# B&R Automation Studio project prjAxis
Automation Studio 6.0.1.7; technology packages: mappMotion 6.0.437033, OpcUaCs 6.0.0

## Configuration Config1

CPU X20CP1686X, AutomationRuntime 6.0.0, Build 11.3.0, Safety 0.0, Vc 6.0.1

### Task classes (Cpu.sw)
```
Cyclic#1 (cycle 2000 us, tolerance 0 us):
  Program <- Program.prg
DataObjects: McAcpSys
NcDataObjects: Capping <- Capping.dob, McDriveLog
Binaries: arsvcreg, udbdef, McAcpDrv, arflatprv, arcoal, FWRules, TCData, McAcpSim, ashwd, Config_1, ashwac, User, sysconf, asfw, arconfig, iomap, Config_3, Config_2, Role
Libraries: runtime, asieccon, powerlnk, astime, fileio, asepl, sys_lib, McBase, MpBase, McAcpAx, McAxis, MpAxis
```

### Hardware
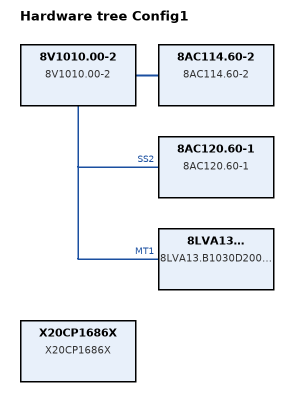
```
8AC114.60-2 : 8AC114.60-2 v2.2.0.0 (NodeNumber=1)  [SS -> 8V1010.00-2.SS1; PLK1 -> X20CP1686X.IF3 [Cable Type=PowerlinkCable, Length=10, Version=1.0.0.3]]
8AC120.60-1 : 8AC120.60-1 v2.2.0.0  [SS -> 8V1010.00-2.SS2]
  PlugInType = Encoder
  McAcoposTypeID = AcoposPlugInConfig
8LVA13.B1030D200-0 : 8LVA13.B1030D200-0 v2.2.0.4  [MT -> 8V1010.00-2.MT1]
  M1/MotorParameters:
    MOTOR_AMB_TEMP_RATED = 40
8V1010.00-2 : 8V1010.00-2 v2.3.0.1
  DriveConfiguration/Module:
    McAcoposTypeID = AcoposConfig
    ActivateACOPOSSimulationOnPLC = 0
    PowerSupply = ETA
  DriveConfiguration/Channel[1]/RealAxis:
    AxisReference = gAxisMaster
    MechanicalElementsIsInvisible = 0
  DriveConfiguration/Channel[1]/RealAxis/MechanicalElements/Gearbox:
    InputIsReadOnly = 0
    Input = 1
    OutputIsReadOnly = 0
    Output = 1
  DriveConfiguration/Channel[1]/RealAxis/MechanicalElements/RotaryToLinearTransformation:
    ReferenceDistanceIsReadOnly = 0
    ReferenceDistance = 1
  DriveConfiguration/Channel[1]/RealAxis/Controller:
    ModeIsReadOnly = 0
    Mode = PositionController
  DriveConfiguration/Channel[1]/RealAxis/Controller/Mode/Position:
    ProportionalGain = 50.0
    IntegrationTime = 0.0
    PredictionTime = 0.0004
    TotalDelayTime = 0.0004
  DriveConfiguration/Channel[1]/RealAxis/Controller/Mode/Speed:
    ProportionalGainIsReadOnly = 0
    ProportionalGain = 2.0
    IntegrationTimeIsReadOnly = 0
    IntegrationTime = 0.0
    FilterTimeIsReadOnly = 0
    FilterTime = 0.0
  DriveConfiguration/Channel[1]/RealAxis/Controller/Mode/LoopFilters:
    LoopFilterXIsReadOnly = 0
    LoopFilter1 = NotUsed
    LoopFilter2 = NotUsed
    LoopFilter3 = NotUsed
  DriveConfiguration/Channel[1]/RealAxis/Homing:
    ModeIsReadOnly = 0
    Mode = Direct
  DriveConfiguration/Channel[1]/RealAxis/Homing/Mode:
    Position = 0.0
    ReferencePulse = NotUsed
  DriveConfiguration/Channel[1]/RealAxis/Homing:
    RestorePositionVariable = 
  DriveConfiguration/Channel[1]/RealAxis/StopReaction:
    QuickstopIsReadOnly = 0
    Quickstop = DecelerationLimit
    DriveErrorIsReadOnly = 0
    DriveError = DecelerationLimit
  DriveConfiguration/Channel[1]/RealAxis/MovementErrorLimits:
    PositionError = 10.0
    VelocityErrorMonitoring = Automatic1
  DriveConfiguration/Channel[1]/RealAxis:
    JerkFilterIsReadOnly = 0
    JerkFilter = NotUsed
    ZeroVibrationFilter = NotUsed
  DriveConfiguration/Channel[1]/RealAxis/DigitalInputs/HomingSwitch:
    SourceIsReadOnly = 0
    Source = X1Ref
    Level = High
  DriveConfiguration/Channel[1]/RealAxis/DigitalInputs/PositiveLimitSwitch:
    Source = X1PosLim
    Level = High
  DriveConfiguration/Channel[1]/RealAxis/DigitalInputs/NegativeLimitSwitch:
    Source = X1NegLim
    Level = High
  DriveConfiguration/Channel[1]/RealAxis/DigitalInputs/Trigger1:
    Source = X1Trigger1
    Level = High
  DriveConfiguration/Channel[1]/RealAxis/DigitalInputs/Trigger2:
    Source = X1Trigger2
    Level = High
  DriveConfiguration/Channel[1]/RealAxis/DigitalInputs/Quickstop:
    Input = Trigger2
  DriveConfiguration/Channel[1]/RealAxis/Simulation:
    SimulationModeOnPLC = CompleteControlledSystem
  DriveConfiguration/Channel[1]/RealAxis/Simulation/SimulationModeOnPLC:
    LoadModel = OneMassBasedOnMotorParameters
  DriveConfiguration/Channel[1]/RealAxis/Simulation/SimulationModeOnPLC/LoadModel:
    AdditiveLoadParID = 0
  DriveConfiguration/Channel[1]/RealAxis/Simulation:
    SimulationModeOnACOPOS = NotUsed
  DriveConfiguration/Channel[1]:
    VirtualAxis = Used
  DriveConfiguration/Channel[1]/VirtualAxis:
    AxisReference = gAxisSlave
  DriveConfiguration/Channel[1]/VirtualAxis/Homing:
    Mode = Direct
  DriveConfiguration/Channel[1]/VirtualAxis/Homing/Mode:
    Position = 0.0
  DriveConfiguration/Channel[1]/VirtualAxis/Homing:
    RestorePositionVariable = 
  DriveConfiguration/Channel[1]/VirtualAxis:
    JerkFilterIsReadOnly = 0
    JerkFilter = NotUsed
    ZeroVibrationFilter = NotUsed
  DriveConfiguration/Channel[1]:
    ExternalEncoderAxis = NotUsed
X20CP1686X : X20CP1686X v1.8.2.0
  Connector IF2:
    ActivateDevice = 1
  Connector IF3:
    CycleTime = 2000
  ConfigurationID = prjAxis_Config1
  TimerDeviceType = EPLX2X
  TimerDevice = X20CP1686X.IF3
  TaskClassIdleTime = 2000
  Cyclic1Duration = 2000
  Cyclic1Tolerance = 0
  FileDevice1
  FileDeviceName1 = USER
  FileDevicePath1 = USER_PATH
  ActivateFtpServer = 1
```

### Config_1.axis - X20CP1686X/mappMotion/Config_1.axis
```
Element gAxisSlave (Type=axis)
  BaseTypeIsReadOnly = 0
  BaseType = RotaryPeriodic
    MeasurementUnitIsReadOnly = 0
    MeasurementUnit = 17476
    MeasurementResolutionIsReadOnly = 0
    MeasurementResolution = 0.01
    CountDirectionIsReadOnly = 0
    CountDirection = Standard
    PeriodSettings:
      Period = 360.0
  MovementLimitsIsReadOnly = 0
  MovementLimits = Internal
    Position:
      LowerLimitMin = -1.79769313486231E308
      UpperLimitMax = 1.79769313486231E308
      LowerLimit = -1000.0
      UpperLimit = 1000.0
    VelocityIsReadOnly = 0
    Velocity:
      VelocityMax = 3.4E38
      Velocity = 720
    AccelerationIsReadOnly = 0
    Acceleration:
      AccelerationMax = 3.4E38
      Acceleration = 3600
    DecelerationIsReadOnly = 0
    Deceleration:
      DecelerationMax = 3.4E38
      Deceleration = 3600
  Alarms = None
Element gAxisMaster (Type=axis)
  BaseTypeIsReadOnly = 0
  BaseType = RotaryPeriodic
    MeasurementUnitIsReadOnly = 0
    MeasurementUnit = 17476
    MeasurementResolutionIsReadOnly = 0
    MeasurementResolution = 0.01
    CountDirectionIsReadOnly = 0
    CountDirection = Standard
    PeriodSettings:
      Period = 360.0
  MovementLimitsIsReadOnly = 0
  MovementLimits = Internal
    Position:
      LowerLimitMin = -1.79769313486231E308
      UpperLimitMax = 1.79769313486231E308
      LowerLimit = -1000.0
      UpperLimit = 1000.0
    VelocityIsReadOnly = 0
    Velocity:
      VelocityMax = 3.4E38
      Velocity = 720
    AccelerationIsReadOnly = 0
    Acceleration:
      AccelerationMax = 3.4E38
      Acceleration = 3600
    DecelerationIsReadOnly = 0
    Deceleration:
      DecelerationMax = 3.4E38
      Deceleration = 3600
  Alarms = None
```

## Logical view

Binary libraries used (declarations not repeated): operator, runtime, astime, AsIecCon, McBase 6.0.437033, MpBase 6.0.7000, McAcpAx 6.0.437033, McAxis 6.0.437033, McAcpPar 6.0.437033, MpAxis 6.0.437033


### Program Logical/Program (IEC)

#### Variables.var
```iecst
VAR
	MpAxisBasic_0 : MpAxisBasic;
	AxisPar : MpAxisBasicParType := (Distance:=30,Velocity:=180,Acceleration:=720,Deceleration:=720);
	MpAxisBasic_1 : MpAxisBasic;
	MpAxisCoupling_0 : MpAxisCoupling;
	CouplingPar : MpAxisCouplingParType := (Gear:=(Acceleration:=720,Deceleration:=720));
	MpAxisCamSequencer_0 : MpAxisCamSequencer;
	SequencerPar : MpAxisCamSequencerParType;
	MpAxisBasic_2 : MpAxisBasic;
	MC_BR_GetAxisLibraryInfo_0 : MC_BR_GetAxisLibraryInfo;
	MC_BR_ProcessParID_AcpAx_0 : MC_BR_ProcessParID_AcpAx;
	processParIdData : McAcpAxProcessParIDType;
	brakeRatedTrq : REAL;
	readMode : BOOL;
	brakeMode : UINT;
END_VAR
```

#### Main.st
```iecst
PROGRAM _INIT
	(* Insert code here *)

	processParIdData.DataType := mcACPAX_PARTYPE_REAL;
	processParIdData.ParID := mcACPPAR_MOTOR_BRAKE_TORQ_RATED;
	processParIdData.VariableAddress := ADR(brakeRatedTrq);

END_PROGRAM

PROGRAM _CYCLIC

	IF readMode THEN
		processParIdData.DataType := mcACPAX_PARTYPE_UINT;

		processParIdData.VariableAddress := ADR(brakeMode);
	ELSE
		processParIdData.DataType := mcACPAX_PARTYPE_REAL;
		processParIdData.ParID := mcACPPAR_MOTOR_BRAKE_TORQ_RATED;
		processParIdData.VariableAddress := ADR(brakeRatedTrq);
	END_IF

	MpAxisBasic_0(MpLink := ADR(gAxisMaster), Enable := TRUE, Parameters := ADR(AxisPar));
	MpAxisBasic_1(MpLink := ADR(gAxisSlave), Enable := TRUE, Parameters := ADR(AxisPar));

	MC_BR_ProcessParID_AcpAx_0(Axis := ADR(gAxisMaster));

END_PROGRAM

PROGRAM _EXIT
	(* Insert code here *)

END_PROGRAM
```

### Data object Logical/Capping (Cam)

#### Cam.cam - Cam for mapp Motion
```
CamProfile (NcSwId=ACP10, MasterAxisVelocity=1, MasterAxisAcceleration=0, DefaultCurveType=Polynomial5, MathematicalNotation=true)
  FixPoint (x=0, IsMathX=true, y=0, IsDefinedDy=false, Dy=0, IsMathDy=true, IsDefinedDdy=false, Ddy=0, IsMathDdy=true, IsDefinedDddy=false, Dddy=0, IsMathDddy=true)
  FixPoint (x=1, IsMathX=true, y=1, IsDefinedDy=false, Dy=0, IsMathDy=true, IsDefinedDdy=false, Ddy=0, IsMathDdy=true, IsDefinedDddy=false, Dddy=0, IsMathDddy=true)
  Synchronline:
    LeftBoundary (IsFix=true, x=0.45, IsMathX=true, y=0.45)
    RightBoundary (IsFix=true, x=0.55, IsMathX=true, y=0.55)
    Gradient (Numerator=1, Denominator=1, IsMath=false, IsFix=false)
  Curve (Type=Polynomial5)
    LeftBoundary (IsDefinedDdy=false, Ddy=0, IsMathDdy=true, IsDefinedDddy=false, Dddy=0, IsMathDddy=true)
    RightBoundary (IsDefinedDdy=false, Ddy=0, IsMathDdy=true, IsDefinedDddy=false, Dddy=0, IsMathDddy=true)
    Spline3 (IsContinuous4Derivative=false, IsDefinedSaddlePoint=false, IsDefinedLineAs2ndSegment=false, IsDefinedSlopeOfLine=false, SlopeOfLine=0, IsMathSlopeOfLine=true)
    Supremum (y=1.7e+308, Dy=1.7e+308, IsMathDy=true, Ddy=1.7e+308, IsMathDdy=true, Dddy=1.7e+308, IsMathDddy=true)
    Infimum (y=-1.7e+308, Dy=-1.7e+308, IsMathDy=true, Ddy=-1.7e+308, IsMathDdy=true, Dddy=-1.7e+308, IsMathDddy=true)
  Curve (Type=Polynomial5)
    LeftBoundary (IsDefinedDdy=false, Ddy=0, IsMathDdy=true, IsDefinedDddy=false, Dddy=0, IsMathDddy=true)
    RightBoundary (IsDefinedDdy=false, Ddy=0, IsMathDdy=true, IsDefinedDddy=false, Dddy=0, IsMathDddy=true)
    Spline3 (IsContinuous4Derivative=false, IsDefinedSaddlePoint=false, IsDefinedLineAs2ndSegment=false, IsDefinedSlopeOfLine=false, SlopeOfLine=0, IsMathSlopeOfLine=true)
    Supremum (y=1.7e+308, Dy=1.7e+308, IsMathDy=true, Ddy=1.7e+308, IsMathDdy=true, Dddy=1.7e+308, IsMathDddy=true)
    Infimum (y=-1.7e+308, Dy=-1.7e+308, IsMathDy=true, Ddy=-1.7e+308, IsMathDdy=true, Dddy=-1.7e+308, IsMathDddy=true)
  Cam (LeftBoundaryIndex=0, RightBoundaryIndex=3)
    Supremum (y=1.7e+308, Dy=1.7e+308, IsMathDy=true, Ddy=1.7e+308, IsMathDdy=true, Dddy=1.7e+308, IsMathDddy=true)
    Infimum (y=-1.7e+308, Dy=-1.7e+308, IsMathDy=true, Ddy=-1.7e+308, IsMathDdy=true, Dddy=1.7e+308, IsMathDddy=true)
  ChartExtensions
```

Listed in the project but not available here: Logical/Global.typ, Logical/Global.var
